FUNCTION_BLOCK FB_Machine_PackML IMPLEMENTS ITF_PackML
VAR
	fbPackML_mem 	: STRUCT_Machine_PackML;
	StepSwitch		: E_State_PackML;
END_VAR

(*
$$$$$$$$\                                                                   $$\       $$$$$$$$\                     $$\                                         $$\                     
$$  _____|                                                                  $$ |      $$  _____|                    \__|                                        \__|                    
$$ |   $$$$$$\   $$$$$$\  $$$$$$$\  $$\  $$\  $$\  $$$$$$\   $$$$$$\   $$$$$$$ |      $$ |      $$$$$$$\   $$$$$$\  $$\ $$$$$$$\   $$$$$$\   $$$$$$\   $$$$$$\  $$\ $$$$$$$\   $$$$$$\  
$$$$$\ \____$$\ $$  __$$\ $$  __$$\ $$ | $$ | $$ |$$  __$$\ $$  __$$\ $$  __$$ |      $$$$$\    $$  __$$\ $$  __$$\ $$ |$$  __$$\ $$  __$$\ $$  __$$\ $$  __$$\ $$ |$$  __$$\ $$  __$$\ 
$$  __|$$$$$$$ |$$ |  \__|$$ |  $$ |$$ | $$ | $$ |$$ /  $$ |$$ /  $$ |$$ /  $$ |      $$  __|   $$ |  $$ |$$ /  $$ |$$ |$$ |  $$ |$$$$$$$$ |$$$$$$$$ |$$ |  \__|$$ |$$ |  $$ |$$ /  $$ |
$$ |  $$  __$$ |$$ |      $$ |  $$ |$$ | $$ | $$ |$$ |  $$ |$$ |  $$ |$$ |  $$ |      $$ |      $$ |  $$ |$$ |  $$ |$$ |$$ |  $$ |$$   ____|$$   ____|$$ |      $$ |$$ |  $$ |$$ |  $$ |
$$ |  \$$$$$$$ |$$ |      $$ |  $$ |\$$$$$\$$$$  |\$$$$$$  |\$$$$$$  |\$$$$$$$ |      $$$$$$$$\ $$ |  $$ |\$$$$$$$ |$$ |$$ |  $$ |\$$$$$$$\ \$$$$$$$\ $$ |      $$ |$$ |  $$ |\$$$$$$$ |
\__|   \_______|\__|      \__|  \__| \_____\____/  \______/  \______/  \_______|      \________|\__|  \__| \____$$ |\__|\__|  \__| \_______| \_______|\__|      \__|\__|  \__| \____$$ |
                                                                                                          $$\   $$ |                                                          $$\   $$ |
                                                                                                          \$$$$$$  |                                                          \$$$$$$  |
                                                                                                           \______/                                                            \______/ 
*)

CASE StepSwitch OF
	E_State_PackML.IDLE 			: 
		//HAPPY FLOW		
		IF fbPackML_mem.Start AND fbPackML_mem.Abort = FALSE THEN
			StepSwitch := E_State_PackML.STARTING;
		END_IF
		
		//EXEPTION HANDLING
		IF fbPackML_mem.Abort THEN
			StepSwitch:= E_State_PackML.ABORTING;
		END_IF
		IF (fbPackML_mem.Stop := TRUE) THEN
			StepSwitch:= E_State_PackML.STOPPING;
		END_IF
	
	E_State_PackML.STARTING 		:
		//HAPPY FLOW		
		IF fbPackML_mem.Starting_SC AND NOT fbPackML_mem.Abort THEN
			StepSwitch:= E_State_PackML.IDLE;
		END_IF
		
		//EXEPTION HANDLING
		IF fbPackML_mem.Abort THEN
			StepSwitch:= E_State_PackML.ABORTING;
		END_IF
		IF fbPackML_mem.Stop THEN
			StepSwitch:= E_State_PackML.STOPPING;
		END_IF
	
	E_State_PackML.EXECUTE 			: 
		//HAPPY FLOW		
		IF (fbPackML_mem.Execute_SC) AND (NOT fbPackML_mem.Abort) THEN
			StepSwitch:= E_State_PackML.IDLE;
		END_IF
		
		IF fbPackML_mem.Hold THEN
			StepSwitch:= E_State_PackML.HOLDING;
		END_IF
		
		IF fbPackML_mem.Suspend THEN
			StepSwitch := E_State_PackML.SUSPENDED;
		END_IF
		
		//EXEPTION HANDLING
		IF fbPackML_mem.Abort THEN
			StepSwitch:= E_State_PackML.ABORTING;
		END_IF
		IF fbPackML_mem.Stop THEN
			StepSwitch:= E_State_PackML.STOPPING;
		END_IF
	
	E_State_PackML.COMPLETE 		:
		//HAPPY FLOW
		StepSwitch:= E_State_PackML.RESETTING;
	
	E_State_PackML.RESETTING 		:
		//HAPPY FLOW		
		IF fbPackML_mem.Resetting_SC AND NOT fbPackML_mem.Abort THEN
			StepSwitch:= E_State_PackML.IDLE;
		END_IF
		
		//EXEPTION HANDLING
		IF fbPackML_mem.Abort THEN
			StepSwitch:= E_State_PackML.ABORTING;
		END_IF
		IF fbPackML_mem.Stop THEN
			StepSwitch:= E_State_PackML.STOPPING;
		END_IF
	
	E_State_PackML.HOLDING 			:
		//HAPPY FLOW		
		IF fbPackML_mem.Holding_SC AND NOT fbPackML_mem.Abort THEN
			StepSwitch:= E_State_PackML.HELD;
		END_IF
		
		//EXEPTION HANDLING
		IF fbPackML_mem.Abort THEN
			StepSwitch:= E_State_PackML.ABORTING;
		END_IF
		IF fbPackML_mem.Stop THEN
			StepSwitch:= E_State_PackML.STOPPING;
		END_IF
		
	
	E_State_PackML.HELD 			:
		//HAPPY FLOW		
		IF fbPackML_mem.Unhold AND NOT fbPackML_mem.Abort THEN
			StepSwitch := E_State_PackML.UNHOLDING;
		END_IF
		
		//EXEPTION HANDLING
		IF fbPackML_mem.Abort THEN
			StepSwitch:= E_State_PackML.ABORTING;
		END_IF
		IF fbPackML_mem.Stop THEN
			StepSwitch:= E_State_PackML.STOPPING;
		END_IF
	
	E_State_PackML.UNHOLDING 		:
		//HAPPY FLOW		
		IF fbPackML_mem.Unholding_SC AND NOT fbPackML_mem.Abort THEN
			StepSwitch:= E_State_PackML.EXECUTE;
		END_IF
		
		//EXEPTION HANDLING
		IF fbPackML_mem.Abort THEN
			StepSwitch:= E_State_PackML.ABORTING;
		END_IF
		IF fbPackML_mem.Stop THEN
			StepSwitch:= E_State_PackML.STOPPING;
		END_IF
	
	E_State_PackML.SUSPENDING 		:
		//HAPPY FLOW		
		IF fbPackML_mem.Suspending_SC AND NOT fbPackML_mem.Abort THEN
			StepSwitch:= E_State_PackML.SUSPENDED;
		END_IF
		
		//EXEPTION HANDLING
		IF fbPackML_mem.Abort THEN
			StepSwitch:= E_State_PackML.ABORTING;
		END_IF
		IF fbPackML_mem.Stop THEN
			StepSwitch:= E_State_PackML.STOPPING;
		END_IF
	
	
	E_State_PackML.SUSPENDED 		:
		//HAPPY FLOW		
		IF fbPackML_mem.Unsuspend AND NOT fbPackML_mem.Abort THEN
			StepSwitch:= E_State_PackML.UNSUSPENDING;
		END_IF
		
		//EXEPTION HANDLING
		IF fbPackML_mem.Abort THEN
			StepSwitch:= E_State_PackML.ABORTING;
		END_IF
		IF fbPackML_mem.Stop THEN
			StepSwitch:= E_State_PackML.STOPPING;
		END_IF
	
	E_State_PackML.UNSUSPENDING 	:
		//HAPPY FLOW		
		IF fbPackML_mem.Unsuspending_SC AND NOT fbPackML_mem.Abort THEN
			StepSwitch:= E_State_PackML.EXECUTE;
		END_IF
		
		//EXEPTION HANDLING
		IF fbPackML_mem.Abort THEN
			StepSwitch:= E_State_PackML.ABORTING;
		END_IF
		IF fbPackML_mem.Stop THEN
			StepSwitch:= E_State_PackML.STOPPING;
		END_IF
	
	E_State_PackML.ABORTED			:
		//HAPPY FLOW		
		IF fbPackML_mem.Clear THEN
			StepSwitch:= E_State_PackML.CLEARING;
		END_IF
	
		
	E_State_PackML.ABORTING			:
		//HAPPY FLOW		
		IF fbPackML_mem.Aborting_SC THEN
			StepSwitch:= E_State_PackML.ABORTED;
		END_IF
	
		
	E_State_PackML.CLEARING 		:
		//HAPPY FLOW		
		IF fbPackML_mem.Clearing_SC THEN
			StepSwitch:= E_State_PackML.STOPPED;
		END_IF
		
		//EXEPTION HANDLING
		IF fbPackML_mem.Abort THEN
			StepSwitch:= E_State_PackML.ABORTING;
		END_IF
		
		
	E_State_PackML.STOPPING 		:
		//HAPPY FLOW
		IF fbPackML_mem.Stopping_SC THEN
			StepSwitch:= E_State_PackML.STOPPED;
		END_IF
		
		//EXEPTION HANDLING
		IF fbPackML_mem.Abort THEN
			StepSwitch:= E_State_PackML.ABORTING;
		END_IF
		
	
	E_State_PackML.STOPPED 			: 
		//HAPPY FLOW
		IF fbPackML_mem.Reset AND NOT fbPackML_mem.Abort THEN
			StepSwitch:= E_State_PackML.RESETTING;
		END_IF
		
		//EXEPTION HANDLING
		IF fbPackML_mem.Abort THEN
			StepSwitch:= E_State_PackML.ABORTING;
		END_IF
		IF fbPackML_mem.Stop THEN
			StepSwitch:= E_State_PackML.STOPPING;
		END_IF
END_CASE

// Set variables FALSE
(*
fbPackML_mem.Abort 			:= FALSE;
fbPackML_mem.Aborting_SC 	:= FALSE;
fbPackML_mem.Clear 			:= FALSE;
fbPackML_mem.Clearing_SC 	:= FALSE;
fbPackML_mem.Execute_SC 	:= FALSE;
fbPackML_mem.Completing_SC	:= FALSE;
fbPackML_mem.Hold 			:= FALSE;
fbPackML_mem.Holding_SC 	:= FALSE;
fbPackML_mem.Reset 			:= FALSE;
fbPackML_mem.Resetting_SC 	:= FALSE;
fbPackML_mem.Start 			:= FALSE;
fbPackML_mem.Starting_SC 	:= FALSE;
fbPackML_mem.Stop 			:= FALSE;
fbPackML_mem.Stopping_SC 	:= FALSE;
fbPackML_mem.Suspend 		:= FALSE;
fbPackML_mem.Suspending_SC 	:= FALSE;
fbPackML_mem.Unhold 		:= FALSE;
fbPackML_mem.Unholding_SC 	:= FALSE;
fbPackML_mem.Unsuspend 		:= FALSE;
*)

{warning 'add method implementation '}
METHOD Abort : BOOL
fbPackML_mem.Abort := TRUE;
END_METHOD

{warning 'add method implementation '}
METHOD Aborting_SC : BOOL
fbPackML_mem.Aborting_SC := TRUE;
END_METHOD

{warning 'add method implementation '}
METHOD Clear : BOOL
fbPackML_mem.Clear := TRUE;
END_METHOD

{warning 'add method implementation '}
METHOD Clearing_SC : BOOL
fbPackML_mem.Clearing_SC := TRUE;
END_METHOD

{warning 'add method implementation '}
METHOD Completing_SC : BOOL
fbPackML_mem.Completing_SC := TRUE;
END_METHOD

{warning 'add method implementation '}
METHOD Execute_SC : BOOL
fbPackML_mem.Execute_SC := TRUE;
END_METHOD

{warning 'add method implementation '}
METHOD FB_init : BOOL
VAR_INPUT
	(* if TRUE, the retain variables are initialized (warm start / cold start)*)
	bInitRetains	: BOOL;
	(* if TRUE, the instance afterwards gets moved into the copy code (online change)*)
	bInCopyCode	: BOOL;
END_VAR
END_METHOD

{warning 'add method implementation '}
METHOD Hold : BOOL
fbPackML_mem.Hold := TRUE;
END_METHOD

{warning 'add method implementation '}
METHOD Holding_SC : BOOL
fbPackML_mem.Holding_SC := TRUE;
END_METHOD

{warning 'add method implementation '}
METHOD Reset : BOOL
fbPackML_mem.Reset := TRUE;
END_METHOD

{warning 'add method implementation '}
METHOD Resetting_SC : BOOL
fbPackML_mem.Resetting_SC := TRUE;
END_METHOD

{warning 'add method implementation '}
METHOD Start : BOOL
fbPackML_mem.Start := TRUE;
END_METHOD

{warning 'add method implementation '}
METHOD Starting_SC : BOOL
fbPackML_mem.Starting_SC := TRUE;
END_METHOD

{warning 'add property implementation'}
PROPERTY State : E_State_PackML
GET
State := StepSwitch;
END_GET
END_PROPERTY

{warning 'add method implementation '}
METHOD Stop : BOOL
fbPackML_mem.Stop := TRUE;
END_METHOD

{warning 'add method implementation '}
METHOD Stopping_SC : BOOL
fbPackML_mem.Stopping_SC := TRUE;
END_METHOD

{warning 'add method implementation '}
METHOD Suspend : BOOL
fbPackML_mem.Suspend := TRUE;
END_METHOD

{warning 'add method implementation '}
METHOD Suspending_SC : BOOL
fbPackML_mem.Suspending_SC := TRUE;
END_METHOD

{warning 'add method implementation '}
METHOD Unhold : BOOL
fbPackML_mem.Unhold := TRUE;
END_METHOD

{warning 'add method implementation '}
METHOD Unholding_SC : BOOL
fbPackML_mem.Unholding_SC := TRUE;
END_METHOD

{warning 'add method implementation '}
METHOD Unsuspend : BOOL
fbPackML_mem.Unsuspend := TRUE;
END_METHOD

METHOD Unsuspending_SC : BOOL
VAR_INPUT
END_VAR
fbPackML_mem.Unsuspending_SC := TRUE;
END_METHOD

{warning 'add method implementation '}
METHOD ZeroAllVar : BOOL
END_METHOD

END_FUNCTION_BLOCK

(* stored: Version 1.1.0.1, ProductVersion 3.1.4024.12
   POU FB_Machine_PackML: Id {0c96e239-3c9c-460c-9e1c-00915d2351c7}, SpecialFunc None
   Folder Methods: Id {2692b1a7-7f53-4742-a95e-2de0b3b517e3}
   Folder Properties: Id {1a61ffe0-5fe7-40e0-82ae-dc75e0516d06}
   Method Abort: Id {f54c4955-f87f-4f9d-b8f3-bf920c7f1f19}
   Method Aborting_SC: Id {04f7a340-07ce-4550-a297-6365020cae9c}
   Method Clear: Id {19faf436-3dfb-49ce-a1be-52e303b50fe9}
   Method Clearing_SC: Id {a3a1e9e6-1ecd-4c49-958e-0c463acf4b66}
   Method Completing_SC: Id {96703eb6-3dea-42f7-844c-ccca82149153}
   Method Execute_SC: Id {552d28e1-2a4a-438d-b0d0-e030a6105e9e}
   Method FB_init: Id {4f45a115-64eb-494d-9b45-2bd5fe373af9}
   Method Hold: Id {53575ac9-3a8d-42b2-afb7-3be0abd62695}
   Method Holding_SC: Id {9ae2709c-0e37-45ea-b5da-84a1eeff22f3}
   Method Reset: Id {cd5e9997-ff8e-4d31-a085-f9181e576959}
   Method Resetting_SC: Id {55276bc5-a368-48f5-b0f2-4f72d7eb9eee}
   Method Start: Id {7bd68d03-d27c-416b-b788-f67971368d7a}
   Method Starting_SC: Id {7d892e21-dd21-4bd9-9552-c6380a0ca1f8}
   Property State: Id {12585bee-b7dc-4602-a0af-aedb1f7976dd}
   Get Get: Id {d588e31c-a050-4e65-bc7f-89fb048b795a}
   Method Stop: Id {05ea9ce5-69ee-49ab-829b-8a4fe1790d84}
   Method Stopping_SC: Id {73f5a823-5695-4d9c-aa3c-396d248d2bc3}
   Method Suspend: Id {483f626d-6ed8-4995-9a57-85f27a1a3922}
   Method Suspending_SC: Id {3e035793-32f7-4a91-9fe9-36c8acdfbdbd}
   Method Unhold: Id {52198064-f668-4596-a17a-dc02abffab17}
   Method Unholding_SC: Id {97c48902-f667-48e2-a7b4-2f07525a1e88}
   Method Unsuspend: Id {3ea7634e-a74f-4336-928c-2f7214c38715}
   Method Unsuspending_SC: Id {a78984c2-4437-4f44-b016-63a7d57366c6}
   Method ZeroAllVar: Id {eff47e16-b2a4-4ccf-ac4e-cb8938c2d680} *)
